(* Schneider Machine Expert - Basic project open close door automatically, file version 2.7.0.0 *)
(* ProjectInformations: Name=New project *)

HARDWARE
  Cpu 0: TM221M16R/G
  EthernetConfiguration: NetworkName=M221, IpAllocationMode=FixedAddress, IpAddress=0.0.0.0, SubnetMask=0.0.0.0
  SerialLineConfiguration: Baud=Baud19200, Parity=ParityEven, DataBits=DataBits8, StopBits=StopBits1, PhysicalMedium=PhysicalMediumRs485, TransmissionMode=TransmissionModeModbusRtu, SlaveId=1, Addressing=SlaveAddressing
  MastTask: UsePeriodScanMode=false, PeriodScan=100
  FastTask: Period=255
  CpuBehavior: StartingMode=StartAsPreviousState, AutoSaveRamOnEeprom=true, WatchdogPeriod=250

SYMBOLS  (address, symbol, comment, settings)
  %M0       MEM
  %M1       TIMER_MEM
  %TM0        [Preset=7, Base=OneSecond]
  %I0.0     STARTING
  %I0.1     STOP
  %I0.2     ADA_ORANG
  %I0.3     LS2
  %I0.4     LS1
  %Q0.0     DOOR_OPEN
  %Q0.1     DOOR_CLOSE

POU New POU
  (* SectionNumber=1 *)

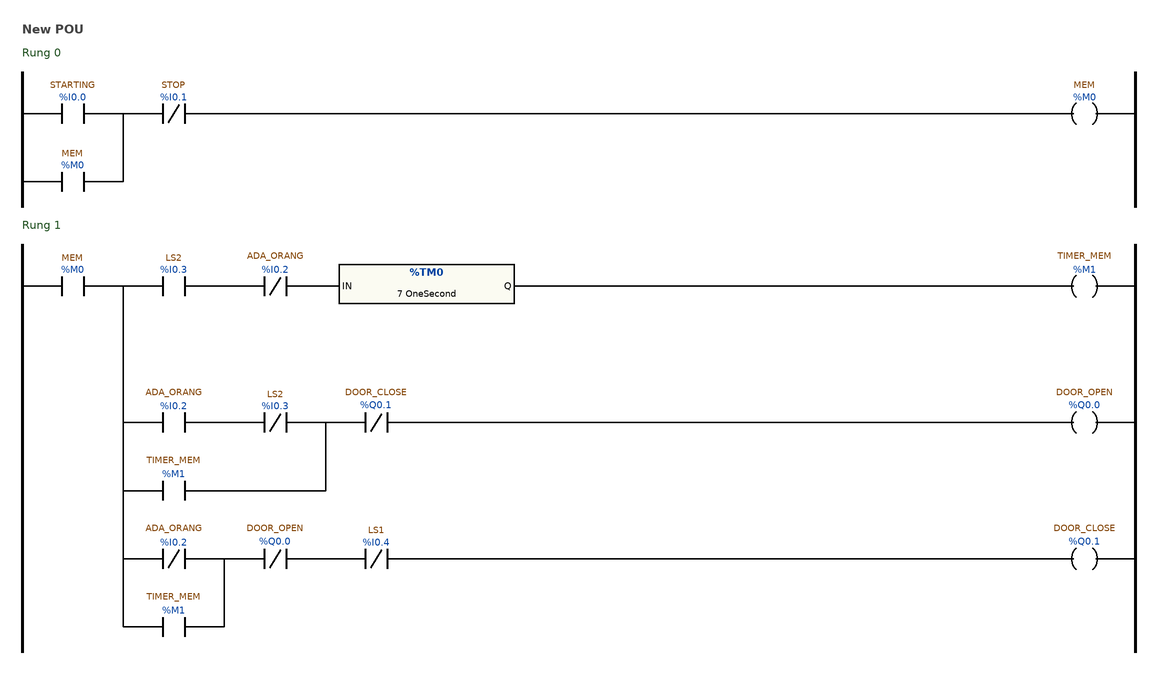

// Rung 0
  LD %I0.0                (* STARTING *)
  OR %M0                  (* MEM *)
  ANDN %I0.1              (* STOP *)
  ST %M0                  (* MEM *)
  // as ST:
  //   MEM := (STARTING OR MEM) AND NOT STOP;

// Rung 1
  LD 1
  MULTIFB
  LD 1
  AND %M0                 (* MEM *)
  ST %MW2009:X0
  BLK %TM0
  LD %MW2009:X0
  AND %I0.3               (* LS2 *)
  ANDN %I0.2              (* ADA_ORANG *)
  IN
  OUT_BLK
  LD Q
  ST %M1                  (* TIMER_MEM *)
  END_BLK
  LD %MW2009:X0
  MPS
  AND( %I0.2              (* ADA_ORANG *)
  ANDN %I0.3              (* LS2 *)
  OR %M1                  (* TIMER_MEM *)
  )
  ANDN %Q0.1              (* DOOR_CLOSE *)
  ST %Q0.0                (* DOOR_OPEN *)
  MPP
  AND(N %I0.2             (* ADA_ORANG *)
  OR %M1                  (* TIMER_MEM *)
  )
  ANDN %Q0.0              (* DOOR_OPEN *)
  ANDN %I0.4              (* LS1 *)
  ST %Q0.1                (* DOOR_CLOSE *)
  MULTIFB
  // as ST:
  //   %TM0(IN := MEM AND LS2 AND NOT ADA_ORANG);
  //   TIMER_MEM := %TM0.Q;
  //   DOOR_OPEN := MEM AND (ADA_ORANG AND NOT LS2 OR TIMER_MEM) AND NOT DOOR_CLOSE;
  //   DOOR_CLOSE := MEM AND (NOT ADA_ORANG OR TIMER_MEM) AND NOT DOOR_OPEN AND NOT LS1;
